// TIA Portal V19 export
VAR_GLOBAL   // PLC tag table "Default tag table"
   EMG_STOP AT %I0.0 : Bool;
   HOOTER_RESET AT %I0.1 : Bool;
   POWER_FAIL AT %I0.2 : Bool;
   "AIR PRESSURE FAIL" AT %I0.3 : Bool;
   "CENTRIFUGAL_PUMP-1_TRIP_(FWD)" AT %I0.4 : Bool;
   "CENTRIFUGAL_PUMP-2_TRIP_(RET)" AT %I0.5 : Bool;
   "FLOW SWITCH-1" AT %I0.6 : Bool;
   "FLOW SWITCH-2" AT %I0.7 : Bool;
   "LEVEL_SWITCH-1" AT %I1.0 : Bool;
   "LEVEL_SWITCH-2" AT %I1.1 : Bool;
   "LEVEL_SWITCH-3" AT %I1.2 : Bool;
   "LEVEL_SWITCH-4" AT %I1.3 : Bool;
   SPARE_DI1 AT %I1.4 : Bool;
   SPARE_DI2 AT %I1.5 : Bool;
   "CENTRIFUGAL_PUMP-1(FWD)" AT %Q0.0 : Bool;
   "CENTRIFUGAL_PUMP-2(RET)" AT %Q0.1 : Bool;
   "DOSING_PUMP-1" AT %Q0.2 : Bool;
   SPARE_DO1 AT %Q0.3 : Bool;
   HOOTER AT %Q0.4 : Bool;
   "PBV-125 PURIFIED WATER VESSEL OUTLET VALVE" AT %Q0.5 : Bool;
   "PBV-126 SOFT WATER VESSEL OUTLET VALVE" AT %Q0.6 : Bool;
   "PBV-127 PW INLET LINE" AT %Q0.7 : Bool;
   "PBV-128 PURIFIED WATER VESSEL–SPRAY BALL INLET LINE" AT %Q1.0 : Bool;
   "PBV-129 SOFT WATER VESSEL INLET LINE" AT %Q1.1 : Bool;
   "LEVEL_SWITCH-10" AT %I8.0 : Bool;
   AIR_PRESSURE_SWITCH AT %I8.1 : Bool;
   "PNEUMATIC_VALVE-7" AT %Q8.0 : Bool;
   "PNEUMATIC_VALVE-8" AT %Q8.1 : Bool;
   "PNEUMATIC_VALVE-9" AT %Q8.2 : Bool;
   "PNEUMATIC_VALVE-10" AT %Q8.3 : Bool;
   "PNEUMATIC_VALVE-11" AT %Q8.4 : Bool;
   "PNEUMATIC_VALVE-12" AT %Q8.5 : Bool;
   "PNEUMATIC_VALVE-13" AT %Q8.6 : Bool;
   "PNEUMATIC_VALVE-14" AT %Q8.7 : Bool;
   "PNEUMATIC_VALVE-15" AT %Q12.0 : Bool;
   "PNEUMATIC_VALVE-16" AT %Q12.1 : Bool;
   "PNEUMATIC_VALVE-17" AT %Q12.2 : Bool;
   "PNEUMATIC_VALVE-18" AT %Q12.3 : Bool;
   "PNEUMATIC_VALVE-19" AT %Q12.4 : Bool;
   CT_SENSOR AT %IW128 : Int;
   TS_SENSOR_1 AT %IW130 : Int;
   TS_SENSOR_2 AT %IW132 : Int;
   "CENTRIFUGAL_PUMP-1_RPM" AT %QW128 : Int;
   "DOSING_PUMP-1(4-20mA)" AT %QW130 : Int;
   System_Byte AT %MB1 : Byte;
   FirstScan AT %M1.0 : Bool;
   DiagStatusUpdate AT %M1.1 : Bool;
   AlwaysTRUE AT %M1.2 : Bool;
   AlwaysFALSE AT %M1.3 : Bool;
   "PNEUMATIC_VALVE-20" AT %Q12.5 : Bool;
   "PNEUMATIC_VALVE-21" AT %Q12.6 : Bool;
   "PNEUMATIC_VALVE-22" AT %Q12.7 : Bool;
   "PZDV-1" AT %Q13.0 : Bool;
   "PZDV-2" AT %Q13.1 : Bool;
   "CIP IN" AT %Q13.2 : Bool;
   "CIP OUT" AT %Q13.3 : Bool;
   "PH NOT ACHIEVED POPUP" AT %M100.0 : Bool;
   "PH ACHIEVED POPUP" AT %M100.1 : Bool;
   ALARM_1 AT %M20.0 : Bool;
   P_TRIG AT %M300.0 : Bool;
   ALARM_2 AT %M20.1 : Bool;
   ALARM_3 AT %M20.2 : Bool;
   ALARM_4 AT %M20.3 : Bool;
   ALARM_5 AT %M20.4 : Bool;
   P_TRIG_1 AT %M300.1 : Bool;
   P_TRIG_2 AT %M300.2 : Bool;
   P_TRIG_3 AT %M300.3 : Bool;
   P_TRIG_4 AT %M300.4 : Bool;
   P_TRIG_5 AT %M300.5 : Bool;
   ALARM_6 AT %M20.5 : Bool;
   ALARM_7 AT %M20.6 : Bool;
   P_TRIG_6 AT %M300.6 : Bool;
   P_TRIG_7 AT %M300.7 : Bool;
   ALARM_8 AT %M20.7 : Bool;
   P_TRIG_8 AT %M301.0 : Bool;
   P_TRIG_9 AT %M301.1 : Bool;
   "RINSE-1_START_POPUP" AT %M2.0 : Bool;
   "RINSE-1 RECIRCULATION_OR_DRAIN" AT %M2.1 : Bool;
   PH_ACHIEVED AT %M2.3 : Bool;
   "RINSE-2_START_POPUP" AT %M2.5 : Bool;
   PH_NOT_ACHIEVED AT %M2.4 : Bool;
   POPUPS AT %MW2 : Word;
   "FRESH CYCLE BIT" AT %M70.0 : Bool;
   "HEATING TEMPERATURE" AT %MD4 : Real;
   "HYSTERSIS ANS" AT %MD8 : Real;
   "HEATING BIT ON" AT %M70.1 : Bool;
   Tag_1 AT %QW96 : Int;
   "PUPM-1_SPEED" AT %MD12 : Real;
   ALARM AT %MW200 : Word;
   "ALAKLI / ACID_START" AT %M2.2 : Bool;
   "RINSE-2_RECIRCULATE_OR_DRAIN" AT %M2.6 : Bool;
   "RINSE-3_RECIRCULATION_OR_DRAIN" AT %M3.0 : Bool;
   FINAL_RINSE_START AT %M3.1 : Bool;
   CONDUCTIVITY_ACHIEVED AT %M3.2 : Bool;
   CONDUCTIVITY_NOT_ACHIEVED_RECIRCULATION_OR_FRESH_CYCLE AT %M3.3 : Bool;
   GOING_TO_FRESH_CYCLE AT %M3.4 : Bool;
   ALARM_9 AT %M21.0 : Bool;
   ERROR AT %M80.0 : Bool;
   "REST TESTYT" AT %M11.0 : Bool;
   PTRIG_10 AT %M11.1 : Bool;
   "RINSE-3_START" AT %M2.7 : Bool;
   ALKALI_LOW_LEVEL_POPUP AT %M3.5 : Bool;
   ACID_LOW_LEVEL_POPUP AT %M3.6 : Bool;
   RESET AT %M0.0 : Bool;
   ALKALI_BIT AT %M0.1 : Bool;
   ACID_BIT AT %M0.2 : Bool;
   "ALAKLI / ACID FRESH CYCLE" AT %M0.3 : Bool;
   "ALKALI/ ACID SELECT_POPUP" AT %M3.7 : Bool;
   "ALKALI / ACID DRAIN_SET" AT %M0.4 : Bool;
   FINAL_RINSE_DRAIN_SET AT %M0.5 : Bool;
   CONDUCTIVITY_ACHIEVED_BIT AT %M0.6 : Bool;
   CONDUCTIVITY_NOT_ACHIEVED_BIT AT %M0.7 : Bool;
   ALARM_10 AT %M21.1 : Bool;
   CYCLE_PAUSE_LSW_FWD AT %M16.0 : Bool;
   CYCLE_PAUSE_LSW_RET AT %M16.1 : Bool;
   AUTO_RESET AT %M16.2 : Bool;
   "RINSE-1_OVER" AT %M17.0 : Bool;
   "ALKALI / ACID_OVER" AT %M17.1 : Bool;
   "RINSE-2_OVER" AT %M17.2 : Bool;
   "FINAL RINSE-1_OVER" AT %M17.3 : Bool;
   "FINAL RINSE-2_OVER" AT %M17.4 : Bool;
   PTRIG_11 AT %M16.3 : Bool;
   PTRIG_12 AT %M16.4 : Bool;
   PTRIG_13 AT %M16.5 : Bool;
   PTRIG_14 AT %M16.6 : Bool;
   PTRIG_15 AT %M16.7 : Bool;
   CYCLE_OVER_ALARM AT %MW17 : Word;
   "CYCLE PAUSE" AT %M19.0 : Bool;
   VACCUME_VALVE_AUTO_BIT AT %M19.1 : Bool;
   N_TRIG AT %M19.2 : Bool;
   P_TRIG_10 AT %M301.2 : Bool;
   ALARM_11 AT %M21.2 : Bool;
   ALARM_12 AT %M21.3 : Bool;
   P_TRIG_11 AT %M301.3 : Bool;
   PTRIG_16 AT %M19.3 : Bool;
   PTRIG_17 AT %M19.4 : Bool;
   N_TRIG1 AT %M19.5 : Bool;
   N_TRIG2 AT %M19.6 : Bool;
   "TRIGGER 1" AT %M19.7 : Bool;
   "SET PRINT BIT" AT %M21.4 : Bool;
   "TAG SET" AT %M21.5 : Bool;
   LENGTH AT %MW22 : Int;
   TRIGGER AT %M70.3 : Bool;
   "EMG TRIG" AT %M24.0 : Bool;
   "AL1 REQ" AT %M24.1 : Bool;
   "AL2 REQ" AT %M24.2 : Bool;
   POWER_TRIG AT %M24.3 : Bool;
   "AL3 REQ" AT %M24.4 : Bool;
   "FWD TRIP_TRIG" AT %M24.5 : Bool;
   "AL4 REQ" AT %M24.6 : Bool;
   "RET TRIP_TRIG" AT %M24.7 : Bool;
   "AL5 REQ" AT %M25.0 : Bool;
   ALKALI_LL_TRIG AT %M25.1 : Bool;
   "AL6 REQ" AT %M25.2 : Bool;
   ACID_LL_TRIG AT %M25.3 : Bool;
   "AL7 REQ" AT %M25.4 : Bool;
   PWT_LL_TRIG AT %M25.5 : Bool;
   "AL8 REQ" AT %M25.6 : Bool;
   SWT_LL_TRIG AT %M25.7 : Bool;
   "AL9 REQ" AT %M26.0 : Bool;
   AIR_TRIG AT %M26.1 : Bool;
   FLS_TRIG AT %M26.2 : Bool;
   "AL10 REQ" AT %M26.3 : Bool;
   "AL11 REQ" AT %M26.4 : Bool;
   RLS_TRIG AT %M26.5 : Bool;
   PRODUCT_NAME AT %IB0 : Char;
   "PROD LENGTH" AT %MW28 : Int;
   "ADD PROD LENGTH" AT %MW30 : Int;
   "EQP LENGTH" AT %MW32 : Int;
   "ADD EQP LENGTH" AT %MW34 : Int;
   "OP LENGTH" AT %MW36 : Int;
   "ADD OP LENGTH" AT %MW38 : Int;
   "BATCH LENGTH" AT %MW40 : Int;
   "BATCH ACTUAL LENGTH" AT %MW42 : Int;
   "RECIPE LENGTH" AT %MW44 : Int;
   "ADD RECIPE LENGTH" AT %MW46 : Int;
   "EMP LENGTH" AT %MW48 : Int;
   "ADD EMP LENGTH" AT %MW50 : Int;
   N_TRIG3 AT %M21.6 : Bool;
   FOOTER AT %M21.7 : Bool;
   P_TRIG20 AT %M26.6 : Bool;
   PNV25 AT %Q13.4 : Bool;
   "SW TANK_START_POPUP" AT %M27.0 : Bool;
   "PW TANK_START_POPUP" AT %M27.1 : Bool;
   "SW TANK_OVER" AT %M27.2 : Bool;
   "PW TANK_OVER" AT %M27.3 : Bool;
   P_TRIG_12 AT %M26.7 : Bool;
   P_TRIG_13 AT %M27.4 : Bool;
   xyz AT %M27.5 : Bool;
   ON AT %M27.6 : Bool;
   ON1 AT %M27.7 : Bool;
   on2 AT %M52.0 : Bool;
   on4 AT %M52.1 : Bool;
   "PASSWORD DB" AT %MW54 : Int;
   "ACK 6MONTH" AT %M52.2 : Bool;
   "ACK 8MONTH" AT %M52.3 : Bool;
   "POPUP FOR 6 MONTH" AT %M52.4 : Bool;
   "POPUP FOR 8 MONTH" AT %M52.5 : Bool;
   "POPUP BIT TRIG" AT %M52.6 : Bool;
   "PBV-130 SOFT WATER VESSEL–SPRAY BALL INLET LINE" AT %Q14.0 : Bool;
   "PBV-131 DOSING PUMP INLET LINE" AT %Q14.1 : Bool;
   "PBV-132 PURIFIED WATER VESSEL OUTLET LINE" AT %Q14.2 : Bool;
   "PBV-133 SOFT WATER VESSEL OUTLET LINE" AT %Q14.3 : Bool;
   "PBV-134 FORWARD PUMP INLET LINE" AT %Q14.4 : Bool;
   "PBV-135 REVERSE PUMP CASING DRAIN" AT %Q14.5 : Bool;
   "PBV-136 FORWARD PUMP RECIRCULATION LINE" AT %Q14.6 : Bool;
   "PBV-137 FORWARD PUMP TO HEAT EXCHANGER LINE" AT %Q14.7 : Bool;
   "PBV-138 PURIFIED WATER DRAIN LINE" AT %Q15.0 : Bool;
   "PAV-139 HEAT EXCHANGER BYPASS DRAIN" AT %Q15.1 : Bool;
   "PBV-140 HEAT EXCHANGER INLET LINE" AT %Q15.2 : Bool;
   "PAV-141 STEAM INLET LINE" AT %Q15.3 : Bool;
   "PBV-142 FORWARD PUMP RECIRCULATION LINE" AT %Q15.4 : Bool;
   "PBV-143 FORWARD PUMP TO VESSEL INLET LINE" AT %Q15.5 : Bool;
   "PBV-144 VESSEL INLET LINE" AT %Q16.0 : Bool;
   "PBV-145 REVERSE PUMP TO VESSEL RECIRCULATION LINE" AT %Q16.1 : Bool;
   "PBV-146 REVERSE PUMP TO DRAIN LINE" AT %Q16.2 : Bool;
   "PBV-147 REVERSE PUMP CASING DRAIN LINE" AT %Q16.3 : Bool;
   "PBV-148 REVERSE PUMP INLET LINE" AT %Q16.4 : Bool;
   "PBV-157 SOFT WATER DRAIN LINE" AT %Q16.5 : Bool;
   "PBV-158 SOFT WATER VENT VALVE" AT %Q16.6 : Bool;
   "PBV-159 PURIFIED VENT VALVE" AT %Q16.7 : Bool;
   "PBV-160 ALKALI VALVE" AT %Q17.0 : Bool;
   "PBV-161 ACID VALVE" AT %Q17.1 : Bool;
   SPARE_DO4 AT %Q17.2 : Bool;
   SPARE_DO5 AT %Q17.3 : Bool;
   SPARE_DO6 AT %Q17.4 : Bool;
   SPARE_DO7 AT %Q17.5 : Bool;
   SPARE_DO8 AT %Q17.6 : Bool;
   SPARE_DO9 AT %Q17.7 : Bool;
   SPARE_DO2 AT %Q15.6 : Bool;
   SPARE_DO3 AT %Q15.7 : Bool;
   PH_SENSOR AT %IW134 : Int;
END_VAR
